FUNCTION_BLOCK BloqueioAtivaDesativa (* Composite Function Block Type *)
  (* Standard: 61499-2 *)
  (* Version 0.0, 02/03/2026, template *)
  PACKAGE Hidryco.HidrycoLib;
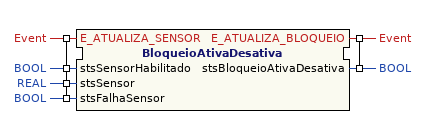
  EVENT_INPUT
    E_ATUALIZA_SENSOR WITH stsSensor, stsFalhaSensor, stsSensorHabilitado;
  END_EVENT
  EVENT_OUTPUT
    E_ATUALIZA_BLOQUEIO WITH stsBloqueioAtivaDesativa;
  END_EVENT
  VAR_INPUT
    stsSensorHabilitado : BOOL;
    stsSensor : REAL;
    stsFalhaSensor : BOOL;
  END_VAR
  VAR_OUTPUT
    stsBloqueioAtivaDesativa : BOOL;
  END_VAR
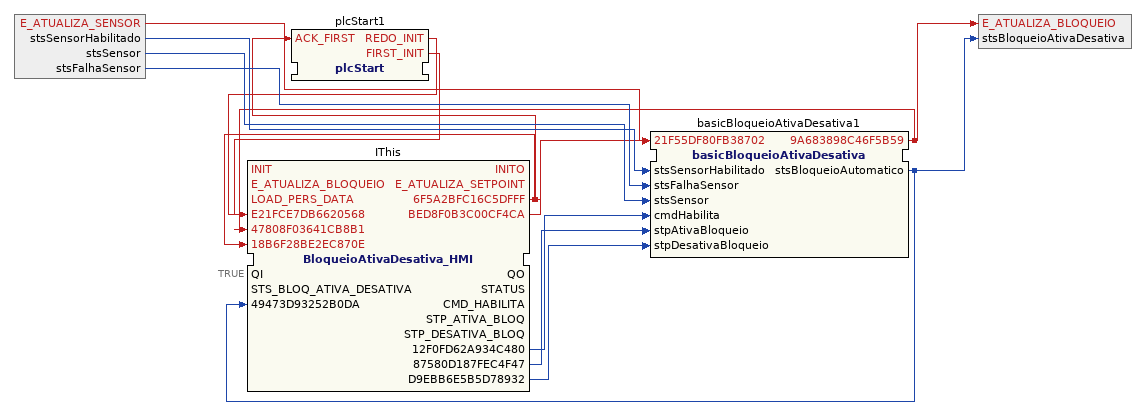
  FBS
    basicBloqueioAtivaDesativa1 : basicBloqueioAtivaDesativa;
    IThis : BloqueioAtivaDesativa_HMI(QI := TRUE);
    plcStart1 : plcStart;
  END_FBS
  EVENT_CONNECTIONS
    plcStart1.REDO_INIT TO IThis.E21FCE7DB6620568;
    plcStart1.FIRST_INIT TO IThis.E21FCE7DB6620568;
    basicBloqueioAtivaDesativa1.9A683898C46F5B59 TO IThis.47808F03641CB8B1;
    IThis.6F5A2BFC16C5DFFF TO IThis.18B6F28BE2EC870E;
    IThis.6F5A2BFC16C5DFFF TO plcStart1.ACK_FIRST;
    IThis.BED8F0B3C00CF4CA TO basicBloqueioAtivaDesativa1.21F55DF80FB38702;
    E_ATUALIZA_SENSOR TO basicBloqueioAtivaDesativa1.21F55DF80FB38702;
    basicBloqueioAtivaDesativa1.9A683898C46F5B59 TO E_ATUALIZA_BLOQUEIO;
  END_CONNECTIONS
  DATA_CONNECTIONS
    stsSensorHabilitado TO basicBloqueioAtivaDesativa1.stsSensorHabilitado;
    stsFalhaSensor TO basicBloqueioAtivaDesativa1.stsFalhaSensor;
    stsSensor TO basicBloqueioAtivaDesativa1.stsSensor;
    basicBloqueioAtivaDesativa1.stsBloqueioAutomatico TO stsBloqueioAtivaDesativa;
    basicBloqueioAtivaDesativa1.stsBloqueioAutomatico TO IThis.49473D93252B0DA;
    IThis.12F0FD62A934C480 TO basicBloqueioAtivaDesativa1.cmdHabilita;
    IThis.87580D187FEC4F47 TO basicBloqueioAtivaDesativa1.stpAtivaBloqueio;
    IThis.D9EBB6E5B5D78932 TO basicBloqueioAtivaDesativa1.stpDesativaBloqueio;
  END_CONNECTIONS
END_FUNCTION_BLOCK
